TYPE EL3433_PM_Outputs :
STRUCT
	{attribute addProperty Name "Index"}
	Index AT %Q* : USINT;
END_STRUCT
END_TYPE

(* stored: Version 1.1.0.1, ProductVersion 3.1.4024.9
   DUT EL3433_PM_Outputs: Id {312056ee-9e35-006a-1969-0d2e6341ea07} *)
